FUNCTION_BLOCK FB_NC_ReadWriteParameters
VAR_INPUT
END_VAR
VAR_OUTPUT
	
		Sts_EncoderOffset					:	REAL;
		Sts_ModuloValue						:	REAL;		

END_VAR
VAR
	
		ReadParameterSet					: 	MC_ReadParameterSet;
		WriteParameter						: 	Tc2_MC2.MC_WriteParameter;
		axisParameterSet	   				:   Tc2_MC2.ST_AxisParameterSet;
		
		StepControl							:	UINT;

END_VAR
VAR_IN_OUT
		Axis								:	Tc2_Mc2.AXIS_REF;
END_VAR

// NC Read / Write Parameters - With standard blocks
// This block is made for inspirational purposes.
// Please make your ovn version that comlies with your / your company´s programming vision
// NOT FINISHED!!!
//-----------------------------------------------------------------------------------------

MC_AxisParameter.AxisEncoderOffset;
MC_AxisParameter.AxisMaximumAcceleration;
MC_AxisParameter.AxisMaximumDeceleration;
MC_AxisParameter.AxisJerk;
MC_AxisParameter.;

// Axis ident
ReadParameterSet(Axis:= Axis,Parameter:= AxisParameterSet);

WriteParameter(Axis:=Axis);


CASE StepControl OF
	
	






END_CASE

END_FUNCTION_BLOCK

(* stored: Version 1.1.0.1, ProductVersion 3.1.4024.14
   POU FB_NC_ReadWriteParameters: Id {3ab1e961-2cf6-4ffb-b70a-671022136d76}, SpecialFunc None *)
